FUNCTION_BLOCK Cylinder EXTENDS CylinderBase
VAR
    {attribute addProperty Name "<#Request move to Home position#>"}
    _moveHomeDefault : CylinderMoveTask(THIS^);
    {attribute addProperty Name "<#Request move to Work position#>"}
    _moveWorkDefault : CylinderMoveTask(THIS^);
    {attribute addProperty Name "<#Request Stop#>"}
    _stopDefault : TcoCore.TcoTask(THIS^);
END_VAR
VAR
    _config : CylinderConfig;
	_status : CylinderStatus;
END_VAR

SUPER^(inoAtHomePos := inoAtHomePos, inoAtWorkPos := inoAtWorkPos, inoToHomePos := inoToHomePos, inoToWorkPos := inoToWorkPos);
// Disables mutually exclusive actions
_moveHomeDefault.Enabled := NOT _moveWorkDefault.Busy;
_moveWorkDefault.Enabled := NOT _moveHomeDefault.Busy;

_moveHomeDefault(PositionSensor := _atHomePos,
    MoveToPositionSignal := _toHomePos,
    InverseSignal := _toWorkPos,
    MaxTimeToReachPosition := _config.TimeToReachHomePosition,
    PositionName := '<#Home#>');
		
_moveWorkDefault(PositionSensor := _atWorkPos,
    MoveToPositionSignal := _toWorkPos,
    InverseSignal := _toHomePos,
    MaxTimeToReachPosition := _config.TimeToReachWorkPosition,
    PositionName := '<#Work#>');

IF (_stopDefault.Execute()) THEN
	_toHomePos := FALSE;
	_toWorkPos := FALSE;
    _moveHomeDefault.Abort();
    _moveWorkDefault.Abort();
    _stopDefault.Abort();
    _moveHomeDefault.Restore();
    _moveWorkDefault.Restore();
    _stopDefault.Restore();
    _stopDefault.DoneWhen(TRUE);
END_IF

// For further discussion about Status
IF(_moveHomeDefault.Busy) THEN
	_status.ActionDescription := 'Moving to home position';
ELSIF(_moveWorkDefault.Busy) THEN
	_status.ActionDescription := 'Moving to work position';
ELSIF(_stopDefault.Busy) THEN
	_status.ActionDescription := 'Stopping pressure';
ELSE	
	_status.ActionDescription := 'Idle';
END_IF

SUPER^(inoAtHomePos := inoAtHomePos, inoAtWorkPos := inoAtWorkPos, inoToHomePos := inoToHomePos, inoToWorkPos := inoToWorkPos);

(*~
	<docu>
		<summary>
			Gets the configuration of the cylinder. 					
		</summary>			
	</docu>	
~*)
PROPERTY Config : REFERENCE TO CylinderConfig
GET
Config REF= config;
END_GET
END_PROPERTY

(*~
	<docu>
		<summary>
			Gets the `MoveHomeTask` task that controls the moving of the cyclinder in home position. 		
		</summary>			
	</docu>	
~*)
PROPERTY MoveHomeTask : TcoCore.ITcoTask
GET
MoveHomeTask := _moveHomeDefault;
END_GET
END_PROPERTY

(*~
	<docu>
		<summary>
			Gets the `MoveWorkTask` task that controls the moving of the cyclinder into work position. 		
		</summary>			
	</docu>	
~*)
PROPERTY MoveWorkTask : TcoCore.ITcoTask
GET
MoveWorkTask := _moveWorkDefault;
END_GET
END_PROPERTY

PROPERTY Status : REFERENCE TO CylinderStatus
GET
Status REF= _status;
END_GET
END_PROPERTY

(*~
	<docu>
		<summary>
			Gets the `StopTask` task that controls the stopping of the cyclinder. 		
		</summary>			
	</docu>	
~*)
PROPERTY StopTask : TcoCore.ITcoTask
GET
StopTask := _stopDefault;
END_GET
END_PROPERTY

END_FUNCTION_BLOCK

(* stored: Version 1.1.0.1, ProductVersion 3.1.4024.6
   POU Cylinder: Id {fe4e2550-76ec-4019-82bb-e68b2cbe4d49}, SpecialFunc None
   Property Config: Id {4900e490-aca6-01f6-34b5-8e88d5861bd7}
   Get Get: Id {01381d79-df26-0dfc-0b34-6d73c1b5b634}
   Property MoveHomeTask: Id {6c5528f8-8b8f-0e7d-01e4-787b210fe4ca}
   Get Get: Id {5717e4b3-14ff-0743-005a-b365bdc9a2e1}
   Property MoveWorkTask: Id {b7eb0230-cd38-0ac9-3271-cda0637a6c51}
   Get Get: Id {d38ced05-e6e6-0894-2289-cb1e2f89ee7d}
   Property Status: Id {4e25aab9-b7e5-00e7-1126-2a4313a14d92}
   Get Get: Id {a32a112b-8373-0a19-170b-cdfdf4b5b4dd}
   Property StopTask: Id {f45f0198-4c17-0e92-3a52-5cc8984cb39c}
   Get Get: Id {28fe28be-dd9b-0922-165d-691ae597ebf9} *)
